TYPE tyOutputs :
STRUCT
	bGasSolenoidValve:BOOL; 
	bAir:BOOL; 
	bIgniter:BOOL; 
	
END_STRUCT
END_TYPE

(* stored: Version 1.1.0.1
   DUT tyOutputs: Id {10f85482-c327-4748-b61f-6e285528b70a} *)
